(*
SPDX-FileCopyrightText: © 2026 Oleksandr Tiutyk <trofimich@gmail.com>
SPDX-License-Identifier: MIT
License: https://opensource.org/license/mit
*)

{attribute 'qualified_only'}
{attribute 'strict'}
{attribute 'to_string'}
TYPE GENERIC_MEMORY_MANAGEMENT_BEHAVIOR :
(
	CLONE_ORIGINAL_VALUE_AND_OWNS_MEMORY,
	STORE_ORIGINAL_REFERENCE_AND_NOT_OWNS_MEMORY,
	STORE_ORIGINAL_REFERENCE_AND_OWNS_MEMORY
);
END_TYPE

(* stored: Version 1.1.0.1
   DUT GENERIC_MEMORY_MANAGEMENT_BEHAVIOR: Id {f71fed05-2a68-457b-995d-be5861a1f1e3} *)
